{attribute 'GeneratedUsingTerminal: ER1098-0001-0017'}
{attribute addProperty BoxType "ER1098-0001-0017"}
{attribute addProperty Id "EtcSlaveTerminalBaseChannel_1AT %I*Channel_830843C11Channel_2AT %I*Channel_830843C11Channel_3AT %I*Channel_830843C11Channel_4AT %I*Channel_830843C11Channel_5AT %I*Channel_830843C11Channel_6AT %I*Channel_830843C11Channel_7AT %I*Channel_830843C11Channel_8AT %I*Channel_830843C11WcStateAT %I*WcState_9091E0EB2InfoDataAT %I*InfoData_6F19DB2B2"}
{attribute addProperty CRC "1107415211"}
{attribute addProperty Size "12"}
TYPE ER1098_4201D0AB EXTENDS EtcSlaveTerminalBase :
STRUCT
	{attribute addProperty Name "Channel_1"}
	Channel_1 : Channel_830843C1;
	{attribute addProperty Name "Channel_2"}
	Channel_2 : Channel_830843C1;
	{attribute addProperty Name "Channel_3"}
	Channel_3 : Channel_830843C1;
	{attribute addProperty Name "Channel_4"}
	Channel_4 : Channel_830843C1;
	{attribute addProperty Name "Channel_5"}
	Channel_5 : Channel_830843C1;
	{attribute addProperty Name "Channel_6"}
	Channel_6 : Channel_830843C1;
	{attribute addProperty Name "Channel_7"}
	Channel_7 : Channel_830843C1;
	{attribute addProperty Name "Channel_8"}
	Channel_8 : Channel_830843C1;
	{attribute addProperty Name "WcState"}
	WcState : WcState_9091E0EB;
	{attribute addProperty Name "InfoData"}
	InfoData : InfoData_6F19DB2B;
END_STRUCT
END_TYPE

(* stored: Version 1.2.0.0, ProductVersion 3.1.4024.9
   DUT ER1098_4201D0AB: Id {bf3b108a-b118-42b5-8d6c-a69b1682a981} *)
